FUNCTION_BLOCK FB_CleaningProcessStateInit EXTENDS FB_CleaningProcessStateBase
VAR_INPUT
END_VAR
VAR_OUTPUT
END_VAR
VAR
	bL_InitActive : BOOL := TRUE;;
END_VAR

METHOD mProduction : BOOL
VAR_INPUT
END_VAR
//Switch to production mode if no operation active
IF I_MachineStatus.pSafetyOk AND I_MachineStatus.pMachineReady AND NOT bL_DevOpActive THEN
	I_ParentCallback.mChangeState(EN_Cleaning_State.Production);
END_IF
END_METHOD

METHOD mService : BOOL
VAR_INPUT
END_VAR
//Switch to service mode
IF NOT bL_DevOpActive THEN
	I_ParentCallback.mChangeState(EN_Cleaning_State.Service);
END_IF
END_METHOD

METHOD mStateAction
VAR_INPUT
END_VAR

VAR
	sL_DeviceStatus : ST_CLEANING_DEV_STATUS;
END_VAR
sL_DeviceStatus := I_ParentCallback.pDeviceStatus;

//If safety ok try to reference axes
IF I_MachineStatus.pSafetyOk AND I_MachineStatus.pMachineReady AND NOT bL_DevOpActive THEN
	//Set mode and start process when successful
	bL_DevOpActive := I_ParentCallback.mSetMode(EN_CLEANING_OP.eOPSTARTUP);
END_IF

IF bL_DevOpActive THEN
	mDevOp();	
END_IF

//If all axes referenced go to service mode
IF sL_DeviceStatus.bError THEN
	I_ParentCallback.mChangeState(EN_Cleaning_State.Error);
ELSIF sL_DeviceStatus.bRefKnown AND NOT sL_DeviceStatus.bBusy THEN
	//I_ParentCallback.mChangeState(EN_Cleaning_State.Service);
	I_ParentCallback.mChangeState(EN_Cleaning_State.Capping);

  bL_InitActive    := FALSE;
  SUPER^.pInitDone := TRUE;
END_IF
END_METHOD

PROPERTY pInitDone : BOOL
GET
pInitDone := NOT bL_InitActive;
END_GET
END_PROPERTY

END_FUNCTION_BLOCK

(* stored: Version 1.1.0.1, ProductVersion 3.1.4024.11
   POU FB_CleaningProcessStateInit: Id {a55095e6-860c-4efa-856e-cb8067d8bb0a}, SpecialFunc None
   Method mProduction: Id {35189b17-d1e9-461b-b9d3-b92e546fd14c}
   Method mService: Id {3dc8b5d8-515f-448f-a35b-e96ce5aaca40}
   Method mStateAction: Id {6d503729-6c6e-4f3b-aff2-4647bb02de1d}
   Property pInitDone: Id {b8abe1ef-6c95-448c-a587-42e0a1d74ad8}
   Get Get: Id {c9887c10-2bbb-4c28-a217-59ccce7a9cf1} *)
